// TwinCAT 3 PLC project Example
// ProgramVersion: 3.1.4026.16
// libraries:
//   Tc2_Standard, * (Beckhoff Automation GmbH)
//   Tc2_System, * (Beckhoff Automation GmbH)
//   Tc2_Utilities, * (Beckhoff Automation GmbH)
//   VisuDialogs, * (System)
//   StageCore, * (_)
//   StageUtils, * (_)
// project tree:
//   / GlobalTextList.TcGTLO (not stored), PlcTask.TcTTO (not stored), Visualization Manager.TcVMO (not stored), VISU_TASK.TcTTO
//   Heating/Ctx/ Heating_Ctx_Hmi.TcPOU, Heating_Ctx_Io.TcDUT (not stored), Heating_Ctx_Priv.TcPOU (not stored), Heating_Ctx_States.TcPOU
//   Heating/Ctx/Io/ Heating_Ctx_Io_In.TcDUT, Heating_Ctx_Io_Out.TcDUT
//   Heating/ Heating.TcPOU (not stored), Heating_Ctx.TcPOU (not stored)
//   Heating/Receivers/ Heating_OnRequest.TcPOU
//   Heating/State/ Heating_State.TcPOU, Heating_State_Enabled.TcPOU, Heating_State_Disabled.TcPOU (not stored), Heating_State_Heatup.TcPOU, Heating_State_HeatingRoom.TcPOU (not stored), Heating_State_Safety.TcPOU (not stored), Heating_State_Fault.TcPOU (not stored)
//   MAIN/ CST.TcGVL (not stored), COL.TcGVL, MAIN.TcPOU, MAIN.TcVIS, SIM.TcGVL
//   MAIN/SIM/ SimulationGlobalParameters.TcDUT (not stored), Tick.TcPOU, ValveSim.TcPOU (not stored)
//   Room/Rooms/ ReceptionRoom.TcPOU (not stored), BaseRoom.TcPOU (not stored), StandardRoom.TcPOU
//   Room/ IArgToIRoom.TcPOU, I_Room.TcIO, Room_Ctx.TcPOU
//   Room/Ctx/ Room_Ctx_Hmi.TcPOU (not stored), Room_Ctx_Io.TcDUT, Room_Ctx_Priv.TcPOU, Room_Ctx_States.TcPOU (not stored)
//   Room/Receivers/ Room_OnSystemEvent.TcPOU
//   Room/State/DemandHeating/ Room_State_DemandHeating.TcPOU, Room_State_DemandHeating_Hmi.TcPOU
//   Room/State/LowTemperature/ Room_State_LowTemperature_Hmi.TcPOU, Room_State_LowTemperature.TcPOU
//   Room/State/ _Room_State.TcPOU, Room_State_Idle.TcPOU, Room_State_Fault.TcPOU (not stored), Room_State_Disabled.TcPOU
//   Room/UI/ Room_UiLogic.TcPOU
//   Safety/ Safety.TcPOU (not stored), Safety_Hmi.TcPOU (not stored)
//   _UI/ UI_Heating.TcVIS, UI_Safety.TcVIS (not stored), UI_Room.TcVIS (not stored), UI_Sim.TcVIS (not stored), UI_Temp.TcVIS, UI_Demand.TcVIS
// (motion and I/O tree: see PLC project stageutils)
// real-time tasks:
//   TASK Example: cycle T#10ms, priority 20, ADS port 350
//   TASK Test: cycle T#10ms, priority 21, ADS port 351
//   TASK VISU_TASK: cycle T#200000us, priority 30, ADS port 352

CONFIGURATION Example
    RESOURCE PLC ON TwinCAT3
        TASK VISU_TASK(INTERVAL := T#200000us, PRIORITY := 30);
        PROGRAM VisuElems_Visu_Prg WITH VISU_TASK : VisuElems.Visu_Prg;
    END_RESOURCE
END_CONFIGURATION

// ---- Heating/Ctx/Io/Heating_Ctx_Io_In.TcDUT
TYPE Heating_Ctx_Io_In :
STRUCT
	bPumpOverload	: BOOL;
	bBurnerOverload	: BOOL;
	
	rBoilerTemp		: LREAL;
	rBoilerPressure	: LREAL;
END_STRUCT
END_TYPE

// ---- Heating/Ctx/Io/Heating_Ctx_Io_Out.TcDUT
TYPE Heating_Ctx_Io_Out :
STRUCT
	bPump			: BOOL;
	bBurner			: BOOL;
END_STRUCT
END_TYPE

// ---- Room/Ctx/Room_Ctx_Io.TcDUT
TYPE Room_Ctx_Io :
STRUCT
	bOpenValves			: BOOL;
	
	bValvesOpen			: BOOL;
	bValvesClosed		: BOOL;
END_STRUCT
END_TYPE

// ---- MAIN/COL.TcGVL
{attribute 'qualified_only'}
VAR_GLOBAL CONSTANT
{warning disable C0228}	// Disable warning: No initial value for variable ...
	RED			: RgbColor(255, 0, 0, 255);
	BLACK		: RgbColor(0, 0, 0, 255);
	ORANGE		: RgbColor(255, 160, 0, 255);
	WHITE		: RgbColor(255, 255, 255, 255);
	INVISIBLE	: RgbColor(0, 0, 0, 0);
{warning restore C0228}
END_VAR

// ---- MAIN/SIM.TcGVL
{attribute 'qualified_only'}
VAR_GLOBAL PERSISTENT
	param			: SimulationGlobalParameters;
END_VAR

VAR_GLOBAL
	bTick				: BOOL;	

	rSystemTemperature	: LREAL := 60;
	rSystemPressure		: LREAL := 1;
	bFlow				: BOOL;
END_VAR

// ---- Room/I_Room.TcIO
INTERFACE I_Room EXTENDS I_Arg

METHOD GoFault
VAR_INPUT
	sErrorText		: Str;
END_VAR
END_METHOD

METHOD GoHeat
END_METHOD

METHOD GoIdle
END_METHOD

PROPERTY Id : UDINT
GET
END_GET
END_PROPERTY

PROPERTY IsActive : BOOL
GET
END_GET
END_PROPERTY

PROPERTY IsClosed : BOOL
GET
END_GET
END_PROPERTY

PROPERTY IsOpen : BOOL
GET
END_GET
END_PROPERTY

PROPERTY IsReady : BOOL
GET
END_GET
END_PROPERTY

PROPERTY Timeout : TIME
GET
END_GET
END_PROPERTY

END_INTERFACE

// ---- Heating/Ctx/Heating_Ctx_Hmi.TcPOU
FUNCTION_BLOCK Heating_Ctx_Hmi
VAR_INPUT
	sStatusText				: Str;
	sErrorText				: Str;
	nStatusColor			: Color;
	
	bButton					: BOOL;
	sButtonText				: Str;
	nButtonColor			: Color;	
END_VAR
VAR_OUTPUT PERSISTENT
	rMaxPressure			: LREAL := 2.0; // bar
	rMinPressure			: LREAL := 0.2; // bar
	
	rMaxTemperature			: LREAL := 65.0; // °C
	rStdTemperature			: LREAL := 60.0; // °C
	rMinTemperature			: LREAL := 55.0; // °C
END_VAR

END_FUNCTION_BLOCK

// ---- Heating/Ctx/Heating_Ctx_States.TcPOU
FUNCTION_BLOCK Heating_Ctx_States
VAR_OUTPUT
	iMgr			: I_StateManager;
	
	iSafety			: I_State;
	iFault			: I_State;
	iDisable		: I_State;
	iEnable			: I_State;
	iHeating		: I_State;
	iHeatup			: I_State;
	
END_VAR

END_FUNCTION_BLOCK

// ---- Heating/Receivers/Heating_OnRequest.TcPOU
FUNCTION_BLOCK Heating_OnRequest IMPLEMENTS I_Callable
VAR
	_ctx			: REFERENCE TO Heating_Ctx;
END_VAR

METHOD Call
VAR_INPUT
	iArg				: StageCore.I_Arg;
END_VAR
VAR
	_iRoom				: I_Room;
END_VAR
IF IsOk(IArgToIRoom(iArg, iDest => _iRoom)) THEN
	_ctx.priv.iQueue.Push(_iRoom);
END_IF
END_METHOD

//FB_Init is always available implicitly and it is used primarily for initialization.
//The return value is not evaluated. For a specific influence, you can also declare the
//methods explicitly and provide additional code there with the standard initialization
//code. You can evaluate the return value.
METHOD FB_Init: BOOL
VAR_INPUT
    bInitRetains: BOOL; // TRUE: the retain variables are initialized (reset warm / reset cold)
    bInCopyCode: BOOL;  // TRUE: the instance will be copied to the copy code afterward (online change)

	ctx			: REFERENCE TO Heating_Ctx;   
END_VAR
_ctx REF= ctx;
END_METHOD

END_FUNCTION_BLOCK

// ---- Room/IArgToIRoom.TcPOU
FUNCTION IArgToIRoom : Result
VAR_INPUT
	iSource	: I_Arg;
END_VAR
VAR_OUTPUT
	iDest	: I_Room;
END_VAR

IF iSource = 0 THEN
	IArgToIRoom := Err.Itf0;
	RETURN;
END_IF

IF __QUERYINTERFACE(iSource, iDest) THEN
	IArgToIRoom := Ok;
ELSE
	iDest := 0;
	IArgToIRoom := Err.NoMatch;
END_IF

END_FUNCTION

// ---- Heating/State/Heating_State.TcPOU
FUNCTION_BLOCK ABSTRACT Heating_State EXTENDS State
VAR
	_ctx			: REFERENCE TO Heating_Ctx;
END_VAR

(*FB_Init is always available implicitly and it is used primarily for initialization.
The return value is not evaluated. For a specific influence, you can also declare the
methods explicitly and provide additional code there with the standard initialization
code. You can evaluate the return value.*)
METHOD FB_Init : BOOL
VAR_INPUT
	(* TRUE: the retain variables are initialized (reset warm / reset cold)*)
	bInitRetains	: BOOL;
	(* TRUE: the instance will be copied to the copy code afterward (online change)*)
	bInCopyCode	: BOOL;
	ctx		: REFERENCE TO Heating_Ctx;
END_VAR
_ctx REF= ctx;
END_METHOD

END_FUNCTION_BLOCK

// ---- Heating/State/Heating_State_Enabled.TcPOU
FUNCTION_BLOCK Heating_State_Enabled EXTENDS Heating_State
VAR_INPUT
END_VAR
VAR_OUTPUT
END_VAR
VAR
END_VAR

METHOD PROTECTED OnEntry
_ctx.hmi.sStatusText := 'Heating enabled: Waiting for requests...';
_ctx.hmi.nStatusColor := COL.BLACK.Raw;

_ctx.hmi.sButtonText := 'Press to DISABLE!';
_ctx.hmi.nButtonColor := COL.BLACK.Raw;

_ctx.io.out.bBurner := FALSE;
_ctx.io.out.bPump := FALSE;

IF _ctx.state.iMgr.Current = _ctx.state.iDisable THEN
	_ctx.priv.iOnEnable.Emit();
END_IF
END_METHOD

METHOD PROTECTED OnExecute
VAR
	_iRoomArg		: I_Arg;
END_VAR
IF _ctx.hmi.bButton THEN
	_ctx.hmi.bButton := FALSE;
	_ctx.state.iMgr.Request(_ctx.state.iDisable);
	
ELSIF _ctx.io.in.rBoilerTemp < _ctx.hmi.rMinTemperature THEN
	_ctx.state.iMgr.Request(_ctx.state.iHeatup);
	
ELSIF IsOk(_ctx.priv.iQueue.Pop(_iRoomArg)) THEN
	IF IsOk(IArgToIRoom(_iRoomArg, iDest => _ctx.priv.iActiveRoom)) THEN
		IF _ctx.priv.iActiveRoom.IsActive THEN
			_ctx.state.iMgr.Request(_ctx.state.iHeating);
		END_IF
	ELSE
		_ctx.hmi.sErrorText := 'Room Queue - Incorrect iRoomArg!';
	END_IF
END_IF
END_METHOD

END_FUNCTION_BLOCK

// ---- Heating/State/Heating_State_Heatup.TcPOU
FUNCTION_BLOCK Heating_State_Heatup EXTENDS Heating_State
VAR_INPUT
END_VAR
VAR_OUTPUT
END_VAR
VAR
END_VAR

METHOD PROTECTED CanActivate : BOOL
CanActivate :=  _ctx.state.iMgr.Current = _ctx.state.iEnable;
END_METHOD

METHOD PROTECTED OnEntry
_ctx.hmi.sStatusText := 'Heating enabled: Heating up...';
_ctx.hmi.nStatusColor := COL.BLACK.Raw;

_ctx.hmi.sButtonText := 'Press to DISABLE!';
_ctx.hmi.nButtonColor := COL.BLACK.Raw;

_ctx.io.out.bBurner := TRUE;
_ctx.io.out.bPump := TRUE;
END_METHOD

METHOD PROTECTED OnExecute
IF _ctx.hmi.bButton THEN
	_ctx.hmi.bButton := FALSE;
	_ctx.state.iMgr.Request(_ctx.state.iDisable);
	
ELSIF _ctx.io.in.rBoilerTemp >= _ctx.hmi.rStdTemperature THEN
	_ctx.state.iMgr.Request(_ctx.state.iEnable);
END_IF
END_METHOD

END_FUNCTION_BLOCK

// ---- MAIN/MAIN.TcPOU
PROGRAM MAIN
VAR
	safety				: Safety<CST.MAX_ESTOP>;
	heating				: Heating<CST.MAX_ROOM>;
	
	stdRoom				: ARRAY[1..3] OF StandardRoom;
	reception			: ReceptionRoom;

	dbgInfo				: DebugInfo;
	rtTick				: R_TRIG;
END_VAR

rtTick(CLK :=  Tick(sim.param.nTick), Q => sim.bTick);
sim.bTick := sim.bTick AND sim.param.bToggleSim;

Runtime();

END_PROGRAM

// ---- Room/Rooms/StandardRoom.TcPOU
FUNCTION_BLOCK StandardRoom EXTENDS BaseRoom
VAR_INPUT
	rTemperature	: LREAL := 20.0 + Math.Random();
END_VAR
VAR    	
    // Entity
    _entityExtend	: EntityExtend(_entityStart);
	
    _lowTemperature : Room_State_LowTemperature(_ctx, rTemperature);
    _demand         : Room_State_DemandHeating(_ctx);
   
    _entityEnd2		: EntityEnd;
END_VAR

METHOD Execute
VAR_INPUT
	nPhase: INT;
END_VAR
SUPER^.Execute(nPhase);

// Simulation
IF NOT sim.bTick THEN
	RETURN;
END_IF

IF bInletValve AND bOutletValve THEN
	rTemperature := rTemperature + sim.param.rRoomTemperatureRisePerHeater * Math.Random();
END_IF

rTemperature := rTemperature + sim.param.rRoomTemperaturePassiveDrop * Math.Random();

IF rTemperature < 0 THEN
	rTemperature := 0;
ELSIF rTemperature > 100 THEN
	rTemperature := 100;
END_IF
END_METHOD

END_FUNCTION_BLOCK

// ---- Room/State/LowTemperature/Room_State_LowTemperature.TcPOU
FUNCTION_BLOCK Room_State_LowTemperature EXTENDS _Room_State IMPLEMENTS I_Execute, I_Init
VAR
	_init					: Init(THIS^);
	_exe					: Execute(THIS^);
	_hmi					: Room_State_LowTemperature_Hmi;
	_rTemperature			: REFERENCE TO LREAL;
END_VAR

METHOD PROTECTED CanActivate : BOOL
CanActivate := _ctx.state.iMgr.Current = _ctx.state.iIdle;
END_METHOD

METHOD Execute
VAR_INPUT
	nPhase: INT;
END_VAR
VAR
	_iSelf		: I_State := THIS^;
	_strb		: strb;
END_VAR
_strb.Set(_ctx.hmi.sData)
		.Append(' ')
		.Append(Strf.Fmt('%0.2f', F_LReal(_rTemperature)))
		.Append(' degC');

_ctx.hmi.sData := _strb.Read();

IF _ctx.state.iMgr.Current <> _ctx.state.iIdle THEN
	RETURN;
END_IF

IF _ctx.state.iMgr.Current = _iSelf THEN
	RETURN;
END_IF

IF _rTemperature < _hmi.rLowTemperature THEN
	_ctx.state.iMgr.Request(THIS^);
END_IF
END_METHOD

(*FB_Init is always available implicitly and it is used primarily for initialization.
The return value is not evaluated. For a specific influence, you can also declare the
methods explicitly and provide additional code there with the standard initialization
code. You can evaluate the return value.*)
METHOD FB_Init : BOOL
VAR_INPUT
	(* TRUE: the retain variables are initialized (reset warm / reset cold)*)
	bInitRetains	: BOOL;
	(* TRUE: the instance will be copied to the copy code afterward (online change)*)
	bInCopyCode	: BOOL;
	ctx				: REFERENCE TO Room_Ctx;
	rTemperature	: REFERENCE TO LREAL;
END_VAR
_rTemperature REF= rTemperature;
END_METHOD

METHOD Init
VAR_INPUT
	nPhase: INT;
END_VAR
VAR
	i			: Iter(1);
	_iEntity	: I_Entity;
	_iRec		: I_Receiver;
	_r			: Result;
	strb		: Strb;
END_VAR
WHILE IsOk(GetNextEntity(_iEntity)) DO
	IF IsNone(HasTagOption(_iEntity, 'Heating')) THEN
		CONTINUE;
	END_IF
	
	IF IsOk(GetReceiver(_iEntity, '*._onRequest', _iRec)) THEN
		IF IsErr(_ctx.priv.iRequestEvent.Pair(_iRec), nOut => _r) THEN
			DebugMsg(_iRec, strb.Append('Cannot pair _onRequest with this receiver! Error code: ').Append(TO_STRING(_r)).Read());
		END_IF
		
		RETURN;
	END_IF
END_WHILE

DebugMsg(THIS^, strb.Append('Cannot pair _requestEvent with a ').Append('_onRequest').Append('!').Read());
DebugMsg(_iEntity, strb.Append('_onRequest').Append(' not found!').Read());
END_METHOD

METHOD PROTECTED OnEntry
_ctx.io.bOpenValves := FALSE;

_ctx.priv.bActive := TRUE;
_ctx.priv.bReady := FALSE;

_ctx.hmi.sStatusText := 'Heating ON: Low Temperature...';
_ctx.hmi.nStatusColor := COL.BLACK.Raw;

_ctx.hmi.bHideReset := TRUE;

_ctx.priv.iRequestEvent.Emit(_ctx);
END_METHOD

METHOD PROTECTED OnExecute
IF _ctx.hmi.bDisable THEN
	_ctx.state.iMgr.Request(_ctx.state.iDisable);
ELSIF _rTemperature >= _hmi.rHighTemperature THEN
	_ctx.priv.bReady := TRUE;
END_IF
END_METHOD

END_FUNCTION_BLOCK

// ---- Room/State/_Room_State.TcPOU
FUNCTION_BLOCK ABSTRACT _Room_State EXTENDS State
VAR
	_ctx	: REFERENCE TO Room_Ctx;
END_VAR

(*FB_Init is always available implicitly and it is used primarily for initialization.
The return value is not evaluated. For a specific influence, you can also declare the
methods explicitly and provide additional code there with the standard initialization
code. You can evaluate the return value.*)
METHOD FB_Init : BOOL
VAR_INPUT
	(* TRUE: the retain variables are initialized (reset warm / reset cold)*)
	bInitRetains	: BOOL;
	(* TRUE: the instance will be copied to the copy code afterward (online change)*)
	bInCopyCode	: BOOL;
	ctx		: REFERENCE TO Room_Ctx;
END_VAR
_ctx REF= ctx;
END_METHOD

END_FUNCTION_BLOCK

// ---- Room/Room_Ctx.TcPOU
FUNCTION_BLOCK Room_Ctx IMPLEMENTS I_Room
VAR_STAT
	_nNextRoom	: UDINT;
END_VAR
VAR_INPUT
	io			: Room_Ctx_Io;
	hmi			: Room_Ctx_Hmi;
	priv		: Room_Ctx_Priv;
END_VAR
VAR_OUTPUT
	state		: Room_Ctx_States;	
END_VAR

//FB_Init is always available implicitly and it is used primarily for initialization.
//The return value is not evaluated. For a specific influence, you can also declare the
//methods explicitly and provide additional code there with the standard initialization
//code. You can evaluate the return value.
METHOD FB_Init: BOOL
VAR_INPUT
    bInitRetains: BOOL; // TRUE: the retain variables are initialized (reset warm / reset cold)
    bInCopyCode: BOOL;  // TRUE: the instance will be copied to the copy code afterward (online change)
END_VAR
_nNextRoom := _nNextRoom + 1;
hmi.nId := _nNextRoom;
END_METHOD

METHOD GoFault
VAR_INPUT
	sErrorText		: Str;
END_VAR
hmi.sErrorText := sErrorText;
state.iMgr.Request(state.iFault);
END_METHOD

METHOD GoHeat
IF NOT priv.bActive THEN
	RETURN;
END_IF

io.bOpenValves := TRUE;
END_METHOD

METHOD GoIdle
IF NOT priv.bActive THEN
	RETURN;
END_IF

state.iMgr.Request(state.iIdle);
END_METHOD

PROPERTY Id : UDINT
GET
Id := hmi.nId;
END_GET
END_PROPERTY

PROPERTY IsActive : BOOL
GET
IsActive := priv.bActive;
END_GET
END_PROPERTY

PROPERTY IsClosed : BOOL
GET
IsClosed := io.bValvesClosed;
END_GET
END_PROPERTY

PROPERTY IsOpen : BOOL
GET
IsOpen := io.bValvesOpen;
END_GET
END_PROPERTY

PROPERTY IsReady : BOOL
GET
IsReady := priv.bReady;
END_GET
END_PROPERTY

PROPERTY Timeout : TIME
GET
Timeout := UDINT_TO_TIME(hmi.nTimeout * 1000 * 60);
END_GET
END_PROPERTY

END_FUNCTION_BLOCK

// ---- Room/Ctx/Room_Ctx_Priv.TcPOU
FUNCTION_BLOCK Room_Ctx_Priv
VAR_INPUT
	bActive			: BOOL;
	bReady			: BOOL;
	
	iRequestEvent	: I_SignalEmit;
	bPaused			: BOOL;
END_VAR

END_FUNCTION_BLOCK

// ---- Room/State/LowTemperature/Room_State_LowTemperature_Hmi.TcPOU
FUNCTION_BLOCK Room_State_LowTemperature_Hmi
VAR_OUTPUT PERSISTENT
	rHighTemperature	: LREAL := 20.0;
	rLowTemperature 	: LREAL := 19.0;
END_VAR

END_FUNCTION_BLOCK

// ---- Room/State/DemandHeating/Room_State_DemandHeating.TcPOU
FUNCTION_BLOCK Room_State_DemandHeating EXTENDS _Room_State IMPLEMENTS I_Execute
VAR
	_exe				: Execute(THIS^);
	_hmi				: Room_State_DemandHeating_Hmi;
	_tonActive			: TON;
END_VAR

METHOD PROTECTED CanActivate : BOOL
CanActivate := _ctx.state.iMgr.Current = _ctx.state.iIdle;
END_METHOD

METHOD Execute
VAR_INPUT
	nPhase: INT;
END_VAR
VAR
	_iSelf		: I_State := THIS^;
	_strb		: Strb;
END_VAR
_strb.Set(_ctx.hmi.sData)
		.Append(' On: ').Append(strf.SimpleTime(_tonActive.ET, 'S', 'M'));

_ctx.hmi.sData := _strb.Read();

IF _ctx.state.iMgr.Current <> _ctx.state.iIdle THEN
	RETURN;
END_IF

IF _ctx.state.iMgr.Current = _iSelf THEN
	RETURN;
END_IF

IF _hmi.bDemandButton THEN
	_ctx.state.iMgr.Request(THIS^);
END_IF
END_METHOD

METHOD Init
VAR
	i			: Iter(1);
	_iEntity	: I_Entity;
	_iRec		: I_Receiver;
	_r			: Result;
	strb		: Strb;
END_VAR
WHILE IsOk(GetNextEntity(_iEntity)) DO
	IF IsNone(HasTagOption(_iEntity, 'Heating')) THEN
		CONTINUE;
	END_IF
	
	IF IsOk(GetReceiver(_iEntity, '*._onRequest', _iRec)) THEN
		IF IsErr(_ctx.priv.iRequestEvent.Pair(_iRec), nOut => _r) THEN
			DebugMsg(_iRec, strb.Append('Cannot pair _onRequest with this receiver! Error code: ').Append(TO_STRING(_r)).Read());
		END_IF
		
		RETURN;
	END_IF
END_WHILE

DebugMsg(THIS^, strb.Append('Cannot pair _requestEvent with a ').Append('_onRequest').Append('!').Read());
DebugMsg(_iEntity, strb.Append('_onRequest').Append(' not found!').Read());
END_METHOD

METHOD PROTECTED OnEntry
_ctx.io.bOpenValves := FALSE;

_ctx.priv.bActive := TRUE;
_ctx.priv.bReady := FALSE;

_ctx.hmi.sStatusText := 'Heating ON: Scheduled demand...';
_ctx.hmi.nStatusColor := COL.BLACK.Raw;

_ctx.hmi.bHideReset := TRUE;

_tonActive(IN := FALSE);

_ctx.priv.iRequestEvent.Emit(_ctx);
END_METHOD

METHOD PROTECTED OnExecute
_tonActive(IN := _ctx.io.bValvesOpen, PT := UDINT_TO_TIME(_hmi.nActivationTime * 1000));
IF _ctx.hmi.bDisable THEN
	_ctx.state.iMgr.Request(_ctx.state.iDisable);
ELSIF NOT _hmi.bDemandButton THEN
	_ctx.priv.bReady := TRUE;
ELSIF _tonActive.Q THEN
	_ctx.priv.bReady := TRUE;
	_hmi.bDemandButton := FALSE;
END_IF
END_METHOD

METHOD PROTECTED OnExit
VAR_INPUT
END_VAR
_hmi.bDemandButton := FALSE;
END_METHOD

END_FUNCTION_BLOCK

// ---- Room/State/DemandHeating/Room_State_DemandHeating_Hmi.TcPOU
FUNCTION_BLOCK Room_State_DemandHeating_Hmi
VAR_INPUT
	bDemandButton		: BOOL;
END_VAR
VAR_OUTPUT PERSISTENT
	nActivationTime			: UDINT := 30;
END_VAR

END_FUNCTION_BLOCK

// ---- MAIN/SIM/Tick.TcPOU
FUNCTION Tick : BOOL
VAR_INPUT
	nTimeInMs	: ULINT;
	nTaskInMs	: ULINT := 20;
END_VAR

Tick := (GetUnixTime() MOD (nTimeInMs * 10_000)) < (nTaskInMs * 10_000);

END_FUNCTION

// ---- Room/Receivers/Room_OnSystemEvent.TcPOU
FUNCTION_BLOCK Room_OnSystemEvent IMPLEMENTS I_Init, I_Callable
VAR
	_init				: Init(THIS^);
	_onSystemEvent		: Receiver(THIS^);
	
	_bError				: BOOL;
	
	_iResumeEvent		: I_Signal;
	_iPauseEvent		: I_Signal;
	_iEnableEvent		: I_Signal;
	_iDisableEvent		: I_Signal;
	
	_ctx				: REFERENCE TO Room_Ctx;
END_VAR

METHOD PRIVATE _GetSignalAndPair
VAR_INPUT
	iEntity		: I_Entity;
	sToFind		: Str;
END_VAR
VAR_OUTPUT
	iSignal	: I_Signal;
END_VAR
VAR
	_r			: Result;
	strb		: Strb;
END_VAR
CASE GetSignal(iEntity, sToFind, iSignal) OF
	Ok:
		IF IsFail(iSignal.Pair(_onSystemEvent), nOut => _r) THEN
			_bError := TRUE;
			DebugMsg(iSignal, strb.Append('Cannot pair _systemRec with this signal! Error code: ').Append(INT_TO_STRING(_r)).Read());
		END_IF
	ELSE
		_bError := TRUE;
		DebugMsg(THIS^, strb.Append('Cannot pair _systemRec with a ').Append(sToFind).Append('!').Read());
		DebugMsg(iEntity, strb.Append(sToFind).Append(' not found!').Read());
END_CASE
END_METHOD

METHOD Call
VAR_INPUT
	iArg	: StageCore.I_Arg;
END_VAR
VAR
	cmp		: TagCmp;
	_iTag	: I_Tag;
END_VAR
IF _bError THEN
	_ctx.hmi.sErrorText := 'Incorrect receiver initialization!';
	_ctx.state.iMgr.Request(_ctx.state.iFault);
	RETURN;
END_IF

IF IsErr(IArgToITag(iArg, _iTag)) THEN
	_ctx.hmi.sErrorText := 'Incorrect call argument!';
	_ctx.state.iMgr.Request(_ctx.state.iFault);
	RETURN;
END_IF

cmp.Set(_iTag);
IF cmp.Match(_iEnableEvent.Tag).IsTrue() THEN
	IF _ctx.state.iMgr.Current = 0 THEN
		RETURN;
	END_IF

	cmp.Set(_ctx.state.iMgr.Current.Tag);
	IF cmp.Match(_ctx.state.iFault.Tag)
			.Match(_ctx.state.iDisable.Tag)
			.Match(_ctx.state.iIdle.Tag)
			.IsTrue() THEN
			
		RETURN;
	END_IF
	
	_ctx.priv.iRequestEvent.Emit(_ctx);
	
	RETURN;
END_IF
END_METHOD

//FB_Init is always available implicitly and it is used primarily for initialization.
//The return value is not evaluated. For a specific influence, you can also declare the
//methods explicitly and provide additional code there with the standard initialization
//code. You can evaluate the return value.
METHOD FB_Init: BOOL
VAR_INPUT
    bInitRetains: BOOL; // TRUE: the retain variables are initialized (reset warm / reset cold)
    bInCopyCode: BOOL;  // TRUE: the instance will be copied to the copy code afterward (online change)
	
	ctx			: REFERENCE TO Room_Ctx;
END_VAR
_ctx REF= ctx;
END_METHOD

METHOD Init
VAR_INPUT
	nPhase: INT;
END_VAR
VAR
	_iEntity	: I_Entity;
END_VAR
WHILE IsOk(GetNextEntity(_iEntity)) DO
	IF IsFail(HasTagOption(_iEntity, 'Heating')) THEN
		CONTINUE;
	END_IF
	
	_GetSignalAndPair(_iEntity, '*._enableEvent', iSignal => _iEnableEvent);
	
	RETURN;
END_WHILE
END_METHOD

END_FUNCTION_BLOCK

// ---- Room/State/Room_State_Idle.TcPOU
FUNCTION_BLOCK Room_State_Idle EXTENDS _Room_State
VAR_INPUT
END_VAR
VAR_OUTPUT
END_VAR
VAR
END_VAR

METHOD PROTECTED OnEntry
_ctx.io.bOpenValves := FALSE;

_ctx.priv.bActive := FALSE;
_ctx.priv.bReady := FALSE;

_ctx.hmi.sStatusText := 'Heating ON: Idle';
_ctx.hmi.nStatusColor := COL.BLACK.Raw;

_ctx.hmi.bHideReset := TRUE;
END_METHOD

METHOD PROTECTED OnExecute
IF _ctx.hmi.bDisable THEN
	_ctx.state.iMgr.Request(_ctx.state.iDisable);
END_IF
END_METHOD

END_FUNCTION_BLOCK

// ---- Room/State/Room_State_Disabled.TcPOU
FUNCTION_BLOCK Room_State_Disabled EXTENDS _Room_State
VAR_INPUT
END_VAR
VAR_OUTPUT
END_VAR
VAR
END_VAR

METHOD PROTECTED OnEntry
_ctx.io.bOpenValves := FALSE;

_ctx.priv.bActive := FALSE;
_ctx.priv.bReady := FALSE;

_ctx.hmi.sStatusText := 'ROOM DISABLED!';
_ctx.hmi.nStatusColor := COL.RED.Raw;

_ctx.hmi.bHideReset := TRUE;
END_METHOD

METHOD PROTECTED OnExecute
IF NOT _ctx.hmi.bDisable THEN
	_ctx.state.iMgr.Request(_ctx.state.iIdle);
END_IF
END_METHOD

END_FUNCTION_BLOCK

// ---- Room/UI/Room_UiLogic.TcPOU
FUNCTION_BLOCK Room_UiLogic IMPLEMENTS I_Execute
VAR_INPUT
END_VAR
VAR_OUTPUT
END_VAR
VAR
	_exe			: Execute(THIS^);
	_ctx			: REFERENCE TO Room_Ctx;
	
	_bPrvDisable	: BOOL;
END_VAR

METHOD Execute
VAR_INPUT
	nPhase: INT;
END_VAR
IF _bPrvDisable <> _ctx.hmi.bDisable THEN
	_bPrvDisable := _ctx.hmi.bDisable;
	
	IF _ctx.hmi.bDisable THEN
		_ctx.hmi.sDisableText := 'Press to ENABLE!';
	ELSE
		_ctx.hmi.sDisableText := 'Press to DISABLE!';
	END_IF	
END_IF
END_METHOD

//FB_Init is always available implicitly and it is used primarily for initialization.
//The return value is not evaluated. For a specific influence, you can also declare the
//methods explicitly and provide additional code there with the standard initialization
//code. You can evaluate the return value.
METHOD FB_Init: BOOL
VAR_INPUT
    bInitRetains: BOOL; // TRUE: the retain variables are initialized (reset warm / reset cold)
    bInCopyCode: BOOL;  // TRUE: the instance will be copied to the copy code afterward (online change)
	
	ctx			: REFERENCE TO Room_Ctx;
END_VAR
_ctx REF= ctx;

IF _ctx.hmi.bDisable THEN
	_ctx.hmi.sDisableText := 'Press to ENABLE!';
ELSE
	_ctx.hmi.sDisableText := 'Press to DISABLE!';
END_IF
END_METHOD

END_FUNCTION_BLOCK

// ---- MAIN/MAIN.TcVIS
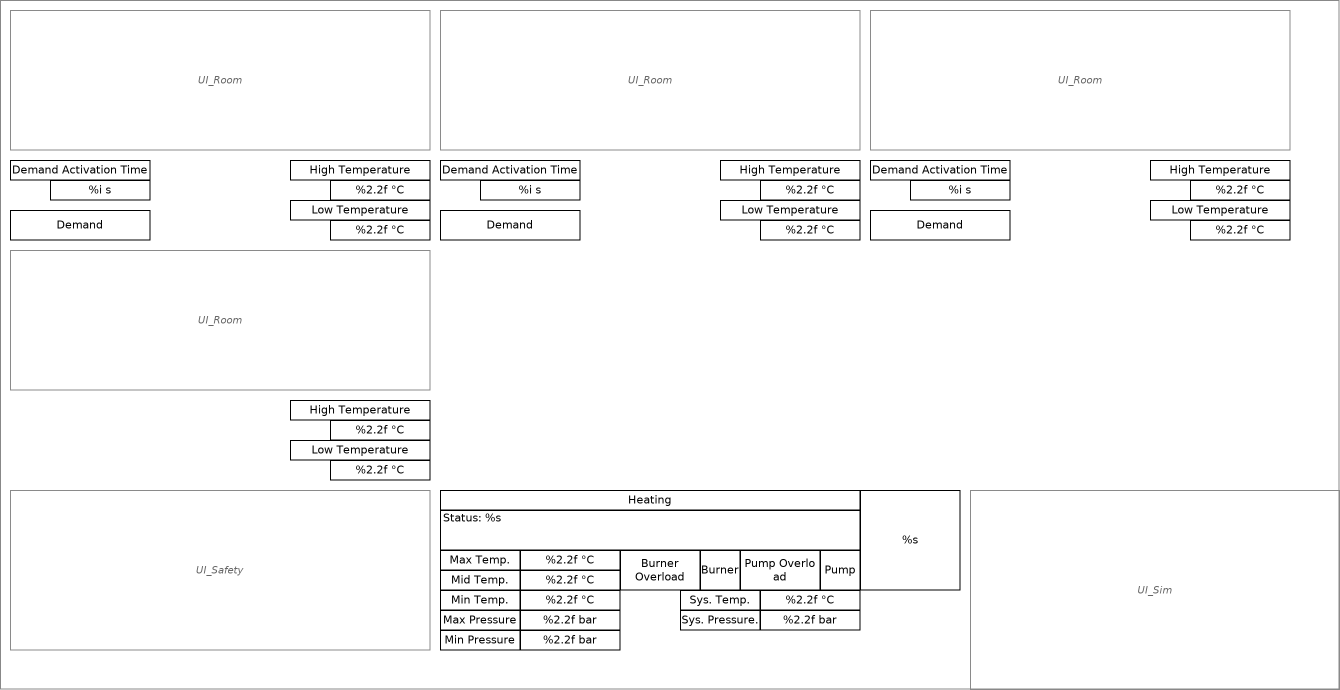
VISUALIZATION MAIN  // 1340x690
    Frame (10,490 420x160)
        shows UI_Safety(pou := MAIN.safety)
    Frame (440,490 520x160)
        shows UI_Heating(pou := MAIN.heating)
    Frame (970,490 370x200)
        shows UI_Sim(param := SIM.param)
    Frame (10,10 420x140)
        shows UI_Room(ctx := MAIN.stdRoom[1]._ctx)
    Frame (290,160 140x80)
        shows UI_Temp(hmi := MAIN.stdRoom[1]._lowTemperature._hmi)
    Frame (10,160 140x80)
        shows UI_Demand(hmi := MAIN.stdRoom[1]._demand._hmi)
    Frame (440,10 420x140)
        shows UI_Room(ctx := MAIN.stdRoom[2]._ctx)
    Frame (720,160 140x80)
        shows UI_Temp(hmi := MAIN.stdRoom[2]._lowTemperature._hmi)
    Frame (440,160 140x80)
        shows UI_Demand(hmi := MAIN.stdRoom[2]._demand._hmi)
    Frame (870,10 420x140)
        shows UI_Room(ctx := MAIN.stdRoom[3]._ctx)
    Frame (1150,160 140x80)
        shows UI_Temp(hmi := MAIN.stdRoom[3]._lowTemperature._hmi)
    Frame (870,160 140x80)
        shows UI_Demand(hmi := MAIN.stdRoom[3]._demand._hmi)
    Frame (10,250 420x140)
        shows UI_Room(ctx := MAIN.reception._ctx)
    Frame (290,400 140x80)
        shows UI_Temp(hmi := MAIN.reception._lowTemperature._hmi)
END_VISUALIZATION

// ---- _UI/UI_Heating.TcVIS
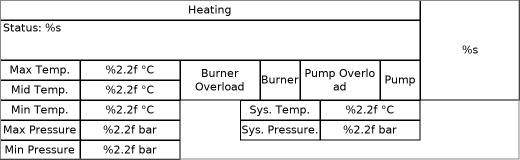
VISUALIZATION UI_Heating  // 520x160
VAR_IN_OUT
	pou			: Heating<CST.MAX_ROOM>;
END_VAR
VAR
END_VAR
    Rectangle (0,0 420x20), "Heating"
    Rectangle (0,20 420x40), "Status: %s", text variable: pou._ctx.hmi.sStatusText
        p55702900: pou._ctx.hmi.nStatusColor
    Rectangle (420,0 100x100), "%s", text variable: pou._ctx.hmi.sButtonText
        p55702900: pou._ctx.hmi.nButtonColor
        toggle pou._ctx.hmi.bButton
    Rectangle (0,60 80x20), "Max Temp."
    Rectangle (0,80 80x20), "Mid Temp."
    Rectangle (0,100 80x20), "Min Temp."
    Rectangle (80,60 100x20), "%2.2f °C", text variable: pou._ctx.hmi.rMaxTemperature
        OnMouseClick: write the text variable via Default
    Rectangle (80,80 100x20), "%2.2f °C", text variable: pou._ctx.hmi.rStdTemperature
        OnMouseClick: write the text variable via Default
    Rectangle (80,100 100x20), "%2.2f °C", text variable: pou._ctx.hmi.rMinTemperature
        OnMouseClick: write the text variable via Default
    Rectangle (0,140 80x20), "Min Pressure"
    Rectangle (0,120 80x20), "Max Pressure"
    Rectangle (80,120 100x20), "%2.2f bar", text variable: pou._ctx.hmi.rMaxPressure
        OnMouseClick: write the text variable via Default
    Rectangle (80,140 100x20), "%2.2f bar", text variable: pou._ctx.hmi.rMinPressure
        OnMouseClick: write the text variable via Default
    Rectangle (380,60 40x40), "Pump", colour toggle: pou.bPump
        toggle pou.bPump
    Rectangle (260,60 40x40), "Burner", colour toggle: pou.bBurner
        toggle pou.bBurner
    Rectangle (300,60 80x40), "Pump Overload", colour toggle: pou.bPumpOverload
        toggle pou.bPumpOverload
    Rectangle (180,60 80x40), "Burner Overload", colour toggle: pou.bBurnerOverload
        toggle pou.bBurnerOverload
    Rectangle (320,120 100x20), "%2.2f bar", text variable: pou.rBoilerPressure
    Rectangle (240,100 80x20), "Sys. Temp."
    Rectangle (240,120 80x20), "Sys. Pressure."
    Rectangle (320,100 100x20), "%2.2f °C", text variable: pou.rBoilerTemp
END_VISUALIZATION

// ---- _UI/UI_Temp.TcVIS
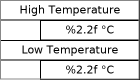
VISUALIZATION UI_Temp  // 140x80
VAR_IN_OUT
	hmi		: Room_State_LowTemperature_Hmi;
END_VAR
    Rectangle (0,40 140x20), "Low Temperature"
    Rectangle (40,60 100x20), "%2.2f °C", text variable: hmi.rLowTemperature
        OnMouseClick: write the text variable via Default
    Rectangle (0,0 140x20), "High Temperature"
    Rectangle (40,20 100x20), "%2.2f °C", text variable: hmi.rHighTemperature
        OnMouseClick: write the text variable via Default
END_VISUALIZATION

// ---- _UI/UI_Demand.TcVIS
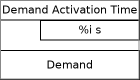
VISUALIZATION UI_Demand  // 140x80
VAR_IN_OUT
	hmi : Room_State_DemandHeating_Hmi;
END_VAR
    Rectangle (40,20 100x20), "%i s", text variable: hmi.nActivationTime
        OnMouseClick: write the text variable via Default
    Rectangle (0,0 140x20), "Demand Activation Time"
    Rectangle (0,50 140x30), "Demand", colour toggle: hmi.bDemandButton
        toggle hmi.bDemandButton
END_VISUALIZATION
